{attribute 'GeneratedUsingTerminal: EL2262-0000-0001'}
{attribute addProperty BoxType "EL2262-0000-0001"}
{attribute addProperty Id "Output0AT %Q*BOOL1"}
{attribute addProperty CRC "2316108"}
{attribute addProperty Size "1"}
TYPE Sample_0023574C :
STRUCT
	{attribute addProperty Name "Output0"}
	Output0 AT %Q* : BOOL;
END_STRUCT
END_TYPE

(* stored: Version 1.2.0.0, ProductVersion 3.1.4024.9
   DUT Sample_0023574C: Id {09eeeebf-e41d-47b6-a512-3f94264fde3e} *)
